PROGRAM MAIN
VAR
	Einlagern: FB_Einlagern;
	iqa_Lager: ARRAY[1..7, 1..12] OF INT;
END_VAR

Einlagern(viqa_Lager := iqa_Lager);

END_PROGRAM

(* stored: Version 1.1.0.1
   POU MAIN: Id {2e83e72e-1aaa-477b-9c8a-106fe183068b}, SpecialFunc None *)
